FUNCTION_BLOCK FB_RealControlBox_ IMPLEMENTS I_ControlBox
VAR_INPUT
END_VAR
VAR_OUTPUT
END_VAR
VAR
END_VAR

{warning 'add method implementation '}
METHOD Joystick
VAR_OUTPUT
	stJoystick	: ST_Joystick;
END_VAR
VAR
	fbJoystickInputScaling : FB_JoystickInputScaling;
	stJoystickInputScaling : ST_JoystickInputScaling;
	//nXInput: INT;
	//nYInput: INT;
END_VAR
//stJoystick := VirtualControlBox.stJOY;
fbJoystickInputScaling(bEnable:=TRUE, 
		nRawInput:=INPUT.nJoyX, 
		stJoystickInputScaling:=stJoystickInputScaling, 
		fNormalizedOutput => ScaledInputs.stJoystick.X);

		
fbJoystickInputScaling(bEnable:=TRUE, 
		nRawInput:=INPUT.nJoyY, 
		stJoystickInputScaling:=stJoystickInputScaling, 
		fNormalizedOutput => ScaledInputs.stJoystick.Y);

ScaledInputs.stJoystick.Topswitch := INPUT.bJoystick;
END_METHOD

{warning 'add method implementation '}
METHOD Mode
VAR_OUTPUT
	eMode	: E_Mode;
END_VAR
VAR
	//eMode : E_Mode;
	bAuto : BOOL;
	bManual : BOOL;
END_VAR
//eMode := VirtualControlBox.eMode;
//OUTPUTS.eMode := eMode;

bAuto := INPUT.bAuto;
bManual := INPUT.bManual;


IF bAuto AND NOT bManual THEN
	eMode := E_Mode.AUTO;
	Working.strMode := 'AUTO';
ELSIF bManual AND NOT bAuto THEN
	eMode := E_Mode.MANUAL;
	Working.strMode := 'MANUAL';
ELSE
	eMode := E_Mode.OFF;
	Working.strMode := 'OFF';
END_IF

Working.eMode := eMode;
END_METHOD

{warning 'add method implementation '}
METHOD Status
VAR
	eStatus : E_Status;
	eMode : E_Mode;
END_VAR
eMode := Working.eMode;
eStatus := Working.eStatus;
CASE eStatus OF
	E_Status.NotReady:
		Working.strStatus := 'NotReady';
		IF eMode <> E_Mode.OFF THEN
			eStatus := E_Status.Ready;
		END_IF
	
	E_Status.Ready:
		Working.strStatus := 'Ready';
		IF eMode = E_Mode.OFF THEN
			eStatus := E_Status.NotReady;
		ELSIF INPUT.bStart THEN
			eStatus := E_Status.Starting;
		END_IF
		
	E_Status.Starting:
		Working.strStatus := 'Starting';
		IF INPUT.bStart AND NOT INPUT.bStop THEN //Add more start conditions?
			eStatus := E_Status.Running;	
		ELSE
			eStatus := E_Status.Ready;
		END_IF
		
	E_Status.Running:	
		Working.strStatus := 'Running';
		IF INPUT.bStop THEN
			eStatus := E_Status.Stopping;
		ELSIF eMode = E_Mode.AUTO THEN
			IF NOT INPUT.bStart THEN // ADD Clock signal
				eStatus := E_Status.Stopping;
			END_IF	
		END_IF
		
	E_Status.Stopping:
		Working.strStatus := 'Stopping';
		//Add stop condition
		eStatus := E_Status.NotReady;
		
	E_Status.Fault:
		Working.strStatus := 'Fault';				
END_CASE

Working.eStatus := eStatus;

//Control Lights
//IF eStatus = E_Status.Running THEN
//	OUTPUTS.bGreenLed := TRUE;
//	OUTPUTS.bEnableCylValve := TRUE;
//	IF ScaledInputs.stJoystick.Topswitch THEN
//		OUTPUTS.bEnableWinchValve := TRUE;
//	ELSE
//		OUTPUTS.bEnableWinchValve := FALSE;
//	END_IF
//ELSE
//	OUTPUTS.bGreenLed := FALSE;
//	OUTPUTS.bEnableCylValve := FALSE;
//	OUTPUTS.bEnableWinchValve := FALSE;
//END_IF

//IF eStatus = E_Status.Stopping OR eStatus = E_Status.Fault THEN
//	OUTPUTS.bRedLed := TRUE;
//ELSE
//	OUTPUTS.bRedLed := FALSE;
//END_IF
END_METHOD

END_FUNCTION_BLOCK

(* stored: Version 1.1.0.1, ProductVersion 3.1.4024.12
   POU FB_RealControlBox_: Id {7323167f-e5d9-471f-b5aa-43d61f819cac}, SpecialFunc None
   Method Joystick: Id {b04946fb-80fe-49f9-8705-7d764bf318a8}
   Method Mode: Id {ce8733aa-10d3-4163-8520-025fe01b837c}
   Method Status: Id {b6e4b7a9-c6a1-4b1e-8a41-7c10228b2ace} *)
